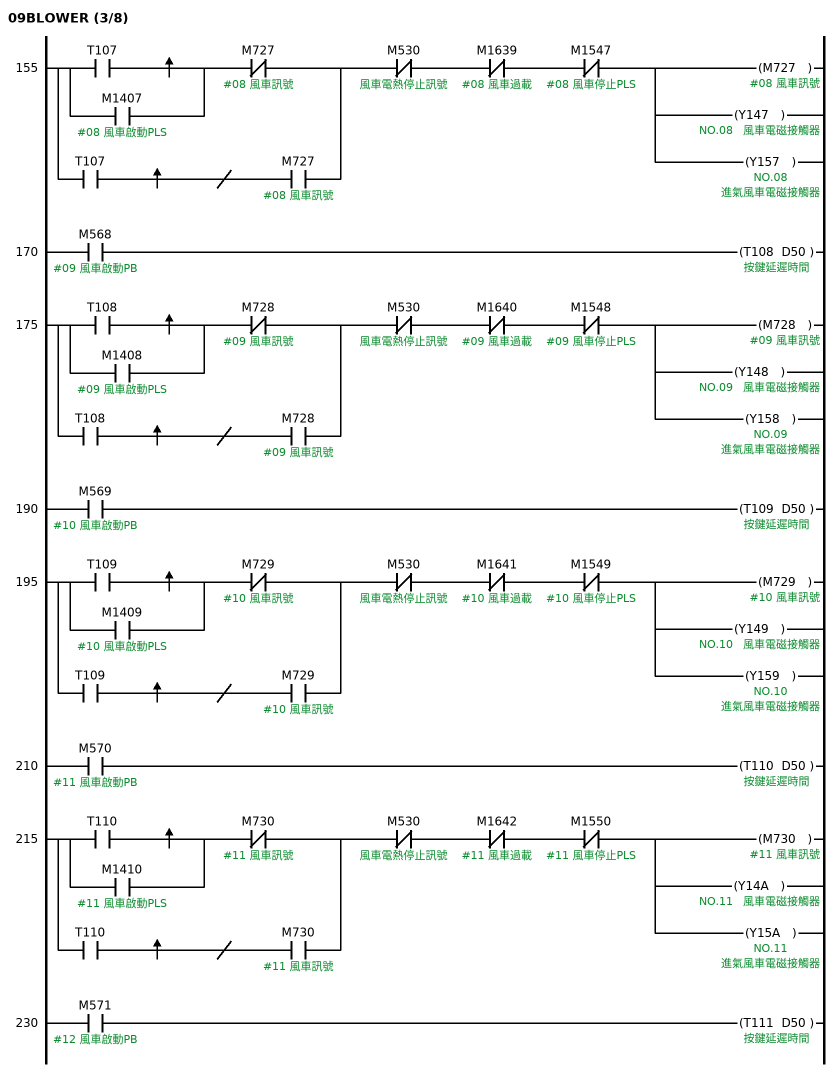
[picture p48: ladder of 09BLOWER, rungs at steps 155 to 230]
155   LD      T107
      MEP
      OR      M1407  ; #08 風車啟動PLS
      ANI     M727  ; #08 風車訊號
      LD      T107
      MEP
      INV
      AND     M727  ; #08 風車訊號
      ORB
      ANI     M530  ; 風車電熱停止訊號
      ANI     M1639  ; #08 風車過載
      ANI     M1547  ; #08 風車停止PLS
      OUT     M727  ; #08 風車訊號
      OUT     Y147  ; NO.08   風車電磁接觸器
      OUT     Y157  ; NO.08   進氣風車電磁接觸器
170   LD      M568  ; #09 風車啟動PB
      OUT     T108 D50  ; 按鍵延遲時間
175   LD      T108
      MEP
      OR      M1408  ; #09 風車啟動PLS
      ANI     M728  ; #09 風車訊號
      LD      T108
      MEP
      INV
      AND     M728  ; #09 風車訊號
      ORB
      ANI     M530  ; 風車電熱停止訊號
      ANI     M1640  ; #09 風車過載
      ANI     M1548  ; #09 風車停止PLS
      OUT     M728  ; #09 風車訊號
      OUT     Y148  ; NO.09   風車電磁接觸器
      OUT     Y158  ; NO.09   進氣風車電磁接觸器
190   LD      M569  ; #10 風車啟動PB
      OUT     T109 D50  ; 按鍵延遲時間
195   LD      T109
      MEP
      OR      M1409  ; #10 風車啟動PLS
      ANI     M729  ; #10 風車訊號
      LD      T109
      MEP
      INV
      AND     M729  ; #10 風車訊號
      ORB
      ANI     M530  ; 風車電熱停止訊號
      ANI     M1641  ; #10 風車過載
      ANI     M1549  ; #10 風車停止PLS
      OUT     M729  ; #10 風車訊號
      OUT     Y149  ; NO.10   風車電磁接觸器
      OUT     Y159  ; NO.10   進氣風車電磁接觸器
210   LD      M570  ; #11 風車啟動PB
      OUT     T110 D50  ; 按鍵延遲時間
215   LD      T110
      MEP
      OR      M1410  ; #11 風車啟動PLS
      ANI     M730  ; #11 風車訊號
      LD      T110
      MEP
      INV
      AND     M730  ; #11 風車訊號
      ORB
      ANI     M530  ; 風車電熱停止訊號
      ANI     M1642  ; #11 風車過載
      ANI     M1550  ; #11 風車停止PLS
      OUT     M730  ; #11 風車訊號
      OUT     Y14A  ; NO.11   風車電磁接觸器
      OUT     Y15A  ; NO.11   進氣風車電磁接觸器
230   LD      M571  ; #12 風車啟動PB
      OUT     T111 D50  ; 按鍵延遲時間
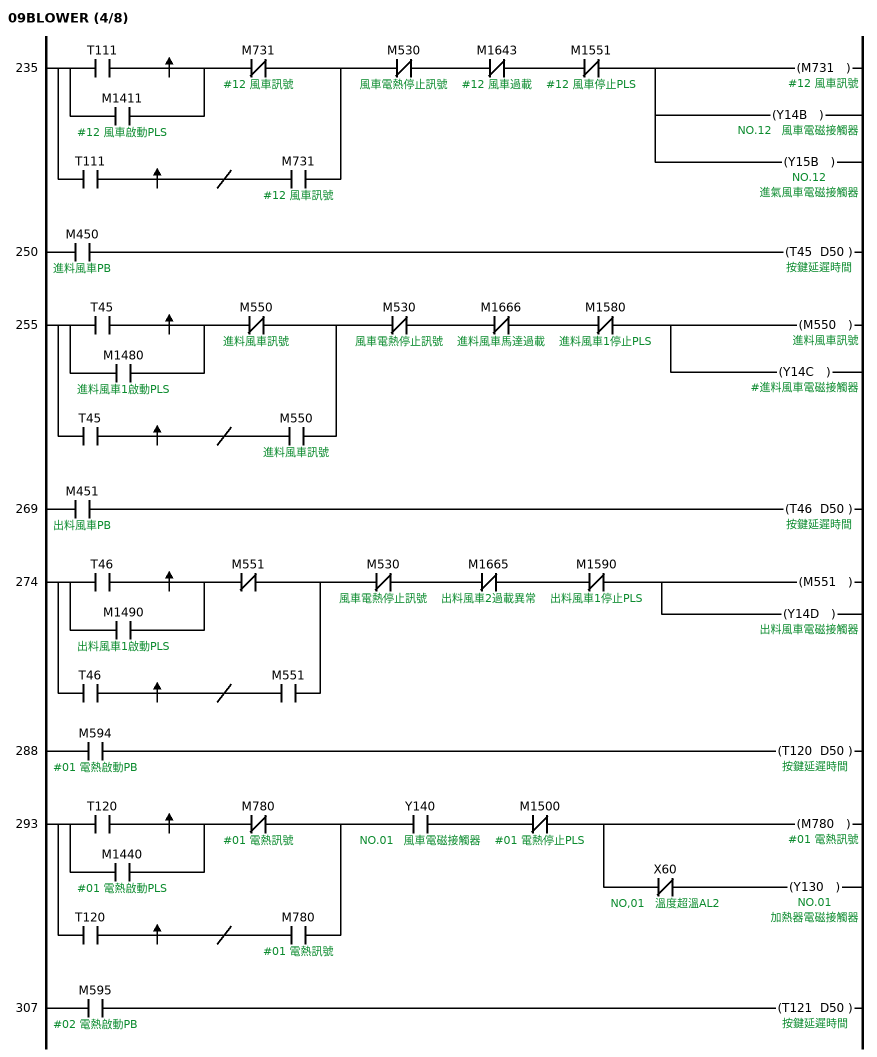
235   LD      T111
      MEP
      OR      M1411  ; #12 風車啟動PLS
      ANI     M731  ; #12 風車訊號
      LD      T111
      MEP
      INV
      AND     M731  ; #12 風車訊號
      ORB
      ANI     M530  ; 風車電熱停止訊號
      ANI     M1643  ; #12 風車過載
      ANI     M1551  ; #12 風車停止PLS
      OUT     M731  ; #12 風車訊號
      OUT     Y14B  ; NO.12   風車電磁接觸器
      OUT     Y15B  ; NO.12   進氣風車電磁接觸器
250   LD      M450  ; 進料風車PB
      OUT     T45 D50  ; 按鍵延遲時間
255   LD      T45
      MEP
      OR      M1480  ; 進料風車1啟動PLS
      ANI     M550  ; 進料風車訊號
      LD      T45
      MEP
      INV
      AND     M550  ; 進料風車訊號
      ORB
      ANI     M530  ; 風車電熱停止訊號
      ANI     M1666  ; 進料風車馬達過載
      ANI     M1580  ; 進料風車1停止PLS
      OUT     M550  ; 進料風車訊號
      OUT     Y14C  ; #進料風車電磁接觸器
269   LD      M451  ; 出料風車PB
      OUT     T46 D50  ; 按鍵延遲時間
274   LD      T46
      MEP
      OR      M1490  ; 出料風車1啟動PLS
      ANI     M551
      LD      T46
      MEP
      INV
      AND     M551
      ORB
      ANI     M530  ; 風車電熱停止訊號
      ANI     M1665  ; 出料風車2過載異常
      ANI     M1590  ; 出料風車1停止PLS
      OUT     M551
      OUT     Y14D  ; 出料風車電磁接觸器
288   LD      M594  ; #01 電熱啟動PB
      OUT     T120 D50  ; 按鍵延遲時間
293   LD      T120
      MEP
      OR      M1440  ; #01 電熱啟動PLS
      ANI     M780  ; #01 電熱訊號
      LD      T120
      MEP
      INV
      AND     M780  ; #01 電熱訊號
      ORB
      AND     Y140  ; NO.01   風車電磁接觸器
      ANI     M1500  ; #01 電熱停止PLS
      OUT     M780  ; #01 電熱訊號
      ANI     X60  ; NO,01   溫度超溫AL2
      OUT     Y130  ; NO.01   加熱器電磁接觸器
307   LD      M595  ; #02 電熱啟動PB
      OUT     T121 D50  ; 按鍵延遲時間
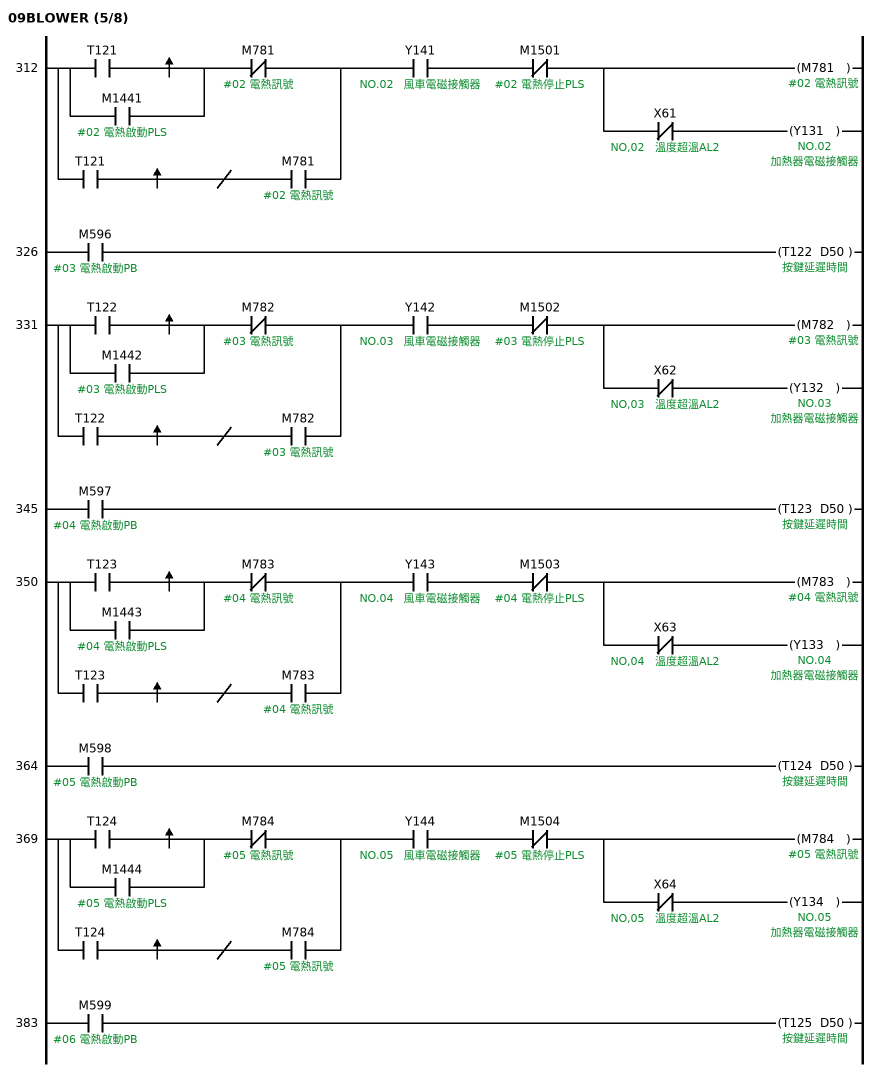
312   LD      T121
      MEP
      OR      M1441  ; #02 電熱啟動PLS
      ANI     M781  ; #02 電熱訊號
      LD      T121
      MEP
      INV
      AND     M781  ; #02 電熱訊號
      ORB
      AND     Y141  ; NO.02   風車電磁接觸器
      ANI     M1501  ; #02 電熱停止PLS
      OUT     M781  ; #02 電熱訊號
      ANI     X61  ; NO,02   溫度超溫AL2
      OUT     Y131  ; NO.02   加熱器電磁接觸器
326   LD      M596  ; #03 電熱啟動PB
      OUT     T122 D50  ; 按鍵延遲時間
331   LD      T122
      MEP
      OR      M1442  ; #03 電熱啟動PLS
      ANI     M782  ; #03 電熱訊號
      LD      T122
      MEP
      INV
      AND     M782  ; #03 電熱訊號
      ORB
      AND     Y142  ; NO.03   風車電磁接觸器
      ANI     M1502  ; #03 電熱停止PLS
      OUT     M782  ; #03 電熱訊號
      ANI     X62  ; NO,03   溫度超溫AL2
      OUT     Y132  ; NO.03   加熱器電磁接觸器
345   LD      M597  ; #04 電熱啟動PB
      OUT     T123 D50  ; 按鍵延遲時間
350   LD      T123
      MEP
      OR      M1443  ; #04 電熱啟動PLS
      ANI     M783  ; #04 電熱訊號
      LD      T123
      MEP
      INV
      AND     M783  ; #04 電熱訊號
      ORB
      AND     Y143  ; NO.04   風車電磁接觸器
      ANI     M1503  ; #04 電熱停止PLS
      OUT     M783  ; #04 電熱訊號
      ANI     X63  ; NO,04   溫度超溫AL2
      OUT     Y133  ; NO.04   加熱器電磁接觸器
364   LD      M598  ; #05 電熱啟動PB
      OUT     T124 D50  ; 按鍵延遲時間
369   LD      T124
      MEP
      OR      M1444  ; #05 電熱啟動PLS
      ANI     M784  ; #05 電熱訊號
      LD      T124
      MEP
      INV
      AND     M784  ; #05 電熱訊號
      ORB
      AND     Y144  ; NO.05   風車電磁接觸器
      ANI     M1504  ; #05 電熱停止PLS
      OUT     M784  ; #05 電熱訊號
      ANI     X64  ; NO,05   溫度超溫AL2
      OUT     Y134  ; NO.05   加熱器電磁接觸器
383   LD      M599  ; #06 電熱啟動PB
      OUT     T125 D50  ; 按鍵延遲時間
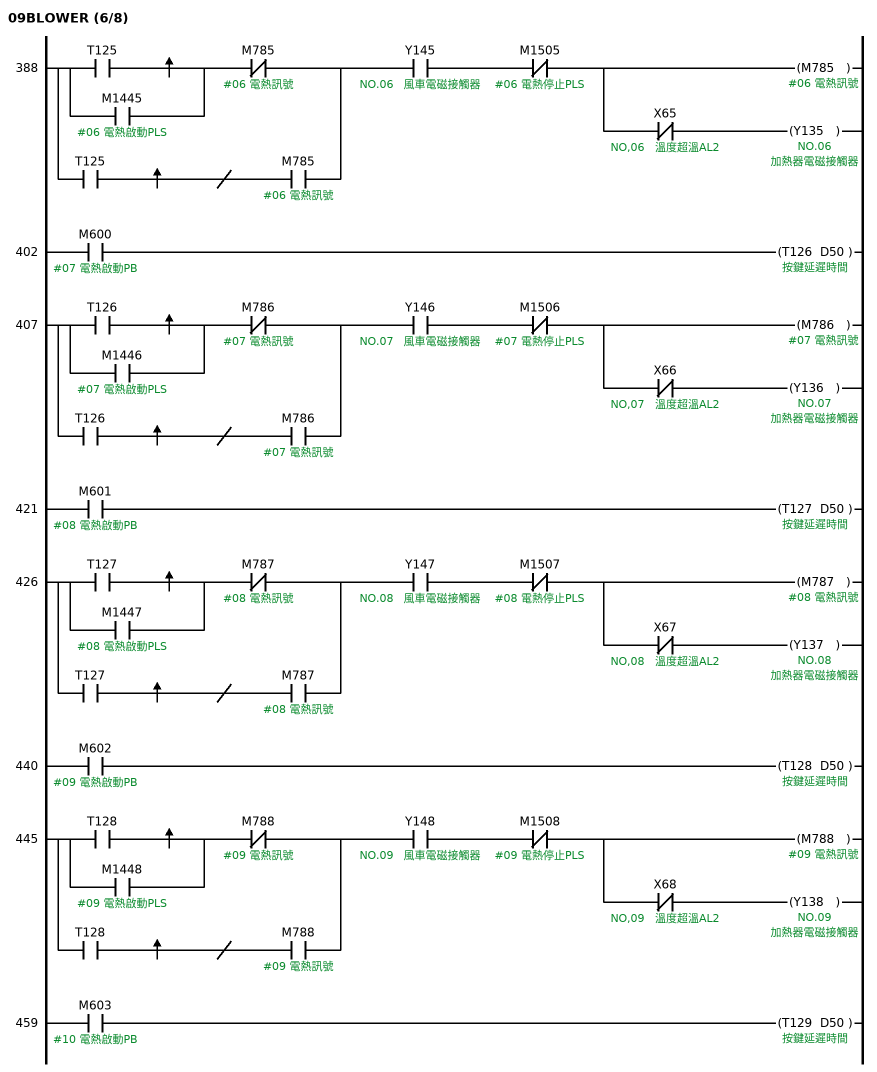
388   LD      T125
      MEP
      OR      M1445  ; #06 電熱啟動PLS
      ANI     M785  ; #06 電熱訊號
      LD      T125
      MEP
      INV
      AND     M785  ; #06 電熱訊號
      ORB
      AND     Y145  ; NO.06   風車電磁接觸器
      ANI     M1505  ; #06 電熱停止PLS
      OUT     M785  ; #06 電熱訊號
      ANI     X65  ; NO,06   溫度超溫AL2
      OUT     Y135  ; NO.06   加熱器電磁接觸器
402   LD      M600  ; #07 電熱啟動PB
      OUT     T126 D50  ; 按鍵延遲時間
407   LD      T126
      MEP
      OR      M1446  ; #07 電熱啟動PLS
      ANI     M786  ; #07 電熱訊號
      LD      T126
      MEP
      INV
      AND     M786  ; #07 電熱訊號
      ORB
      AND     Y146  ; NO.07   風車電磁接觸器
      ANI     M1506  ; #07 電熱停止PLS
      OUT     M786  ; #07 電熱訊號
      ANI     X66  ; NO,07   溫度超溫AL2
      OUT     Y136  ; NO.07   加熱器電磁接觸器
421   LD      M601  ; #08 電熱啟動PB
      OUT     T127 D50  ; 按鍵延遲時間
426   LD      T127
      MEP
      OR      M1447  ; #08 電熱啟動PLS
      ANI     M787  ; #08 電熱訊號
      LD      T127
      MEP
      INV
      AND     M787  ; #08 電熱訊號
      ORB
      AND     Y147  ; NO.08   風車電磁接觸器
      ANI     M1507  ; #08 電熱停止PLS
      OUT     M787  ; #08 電熱訊號
      ANI     X67  ; NO,08   溫度超溫AL2
      OUT     Y137  ; NO.08   加熱器電磁接觸器
440   LD      M602  ; #09 電熱啟動PB
      OUT     T128 D50  ; 按鍵延遲時間
445   LD      T128
      MEP
      OR      M1448  ; #09 電熱啟動PLS
      ANI     M788  ; #09 電熱訊號
      LD      T128
      MEP
      INV
      AND     M788  ; #09 電熱訊號
      ORB
      AND     Y148  ; NO.09   風車電磁接觸器
      ANI     M1508  ; #09 電熱停止PLS
      OUT     M788  ; #09 電熱訊號
      ANI     X68  ; NO,09   溫度超溫AL2
      OUT     Y138  ; NO.09   加熱器電磁接觸器
459   LD      M603  ; #10 電熱啟動PB
      OUT     T129 D50  ; 按鍵延遲時間
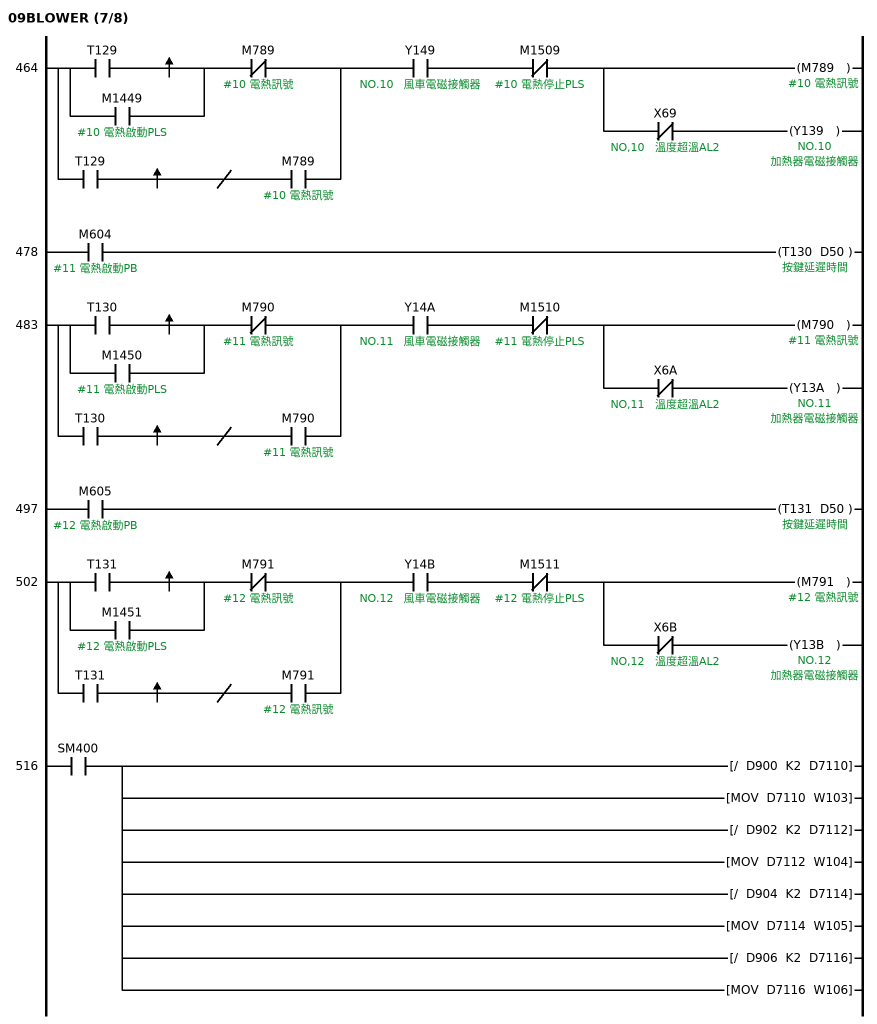
464   LD      T129
      MEP
      OR      M1449  ; #10 電熱啟動PLS
      ANI     M789  ; #10 電熱訊號
      LD      T129
      MEP
      INV
      AND     M789  ; #10 電熱訊號
      ORB
      AND     Y149  ; NO.10   風車電磁接觸器
      ANI     M1509  ; #10 電熱停止PLS
      OUT     M789  ; #10 電熱訊號
      ANI     X69  ; NO,10   溫度超溫AL2
      OUT     Y139  ; NO.10   加熱器電磁接觸器
478   LD      M604  ; #11 電熱啟動PB
      OUT     T130 D50  ; 按鍵延遲時間
483   LD      T130
      MEP
      OR      M1450  ; #11 電熱啟動PLS
      ANI     M790  ; #11 電熱訊號
      LD      T130
      MEP
      INV
      AND     M790  ; #11 電熱訊號
      ORB
      AND     Y14A  ; NO.11   風車電磁接觸器
      ANI     M1510  ; #11 電熱停止PLS
      OUT     M790  ; #11 電熱訊號
      ANI     X6A  ; NO,11   溫度超溫AL2
      OUT     Y13A  ; NO.11   加熱器電磁接觸器
497   LD      M605  ; #12 電熱啟動PB
      OUT     T131 D50  ; 按鍵延遲時間
502   LD      T131
      MEP
      OR      M1451  ; #12 電熱啟動PLS
      ANI     M791  ; #12 電熱訊號
      LD      T131
      MEP
      INV
      AND     M791  ; #12 電熱訊號
      ORB
      AND     Y14B  ; NO.12   風車電磁接觸器
      ANI     M1511  ; #12 電熱停止PLS
      OUT     M791  ; #12 電熱訊號
      ANI     X6B  ; NO,12   溫度超溫AL2
      OUT     Y13B  ; NO.12   加熱器電磁接觸器
516   LD      SM400
      /       D900 K2 D7110
      MOV     D7110 W103
      /       D902 K2 D7112
      MOV     D7112 W104
      /       D904 K2 D7114
      MOV     D7114 W105
      /       D906 K2 D7116
      MOV     D7116 W106
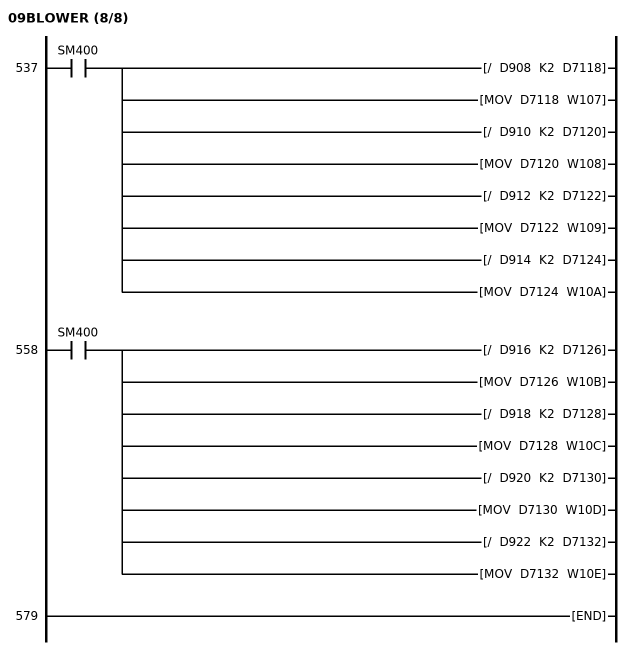
537   LD      SM400
      /       D908 K2 D7118
      MOV     D7118 W107
      /       D910 K2 D7120
      MOV     D7120 W108
      /       D912 K2 D7122
      MOV     D7122 W109
      /       D914 K2 D7124
      MOV     D7124 W10A
558   LD      SM400
      /       D916 K2 D7126
      MOV     D7126 W10B
      /       D918 K2 D7128
      MOV     D7128 W10C
      /       D920 K2 D7130
      MOV     D7130 W10D
      /       D922 K2 D7132
      MOV     D7132 W10E
579   END
END_PROGRAM

PROGRAM 10YIELD
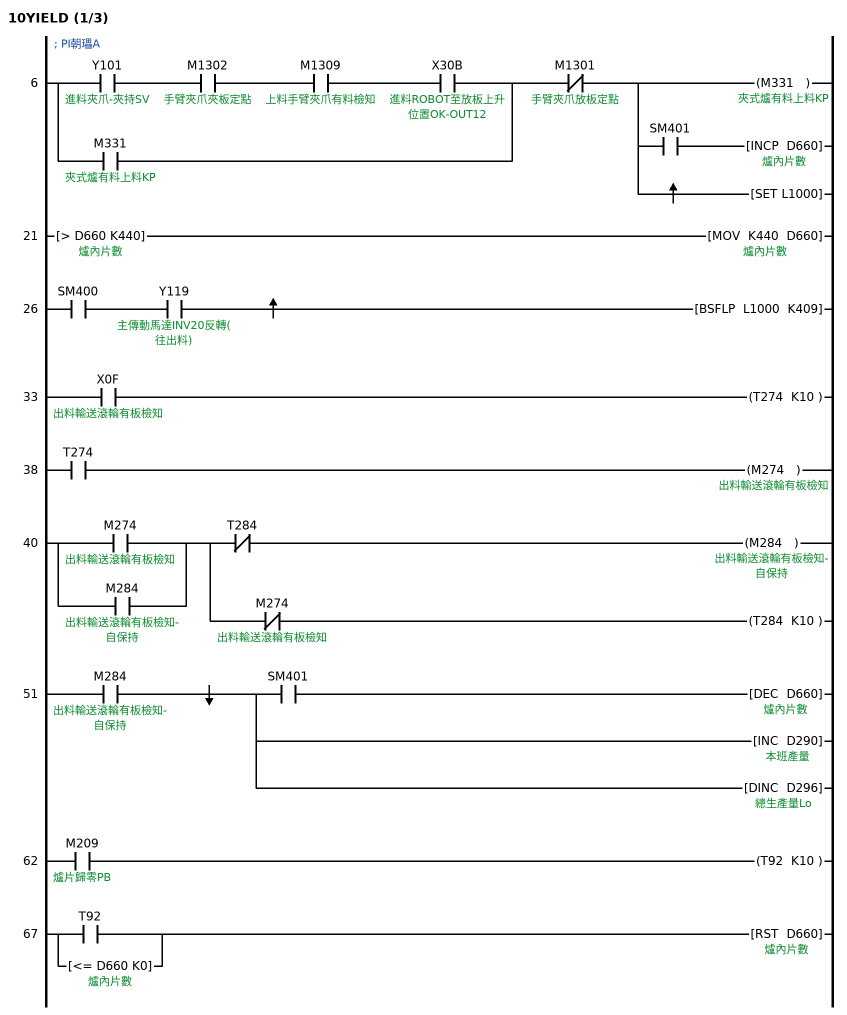
; PI朝瓃Α
6     LD      Y101  ; 進料夾爪-夾持SV
      AND     M1302  ; 手臂夾爪夾板定點
      AND     M1309  ; 上料手臂夾爪有料檢知
      AND     X30B  ; 進料ROBOT至放板上升位置OK-OUT12
      OR      M331  ; 夾式爐有料上料KP
      ANI     M1301  ; 手臂夾爪放板定點
      OUT     M331  ; 夾式爐有料上料KP
      MPS
      AND     SM401
      INCP    D660  ; 爐內片數
      MPP
      MEP
      SET     L1000
21    LD>     D660 K440  ; 爐內片數
      MOV     K440 D660
26    LD      SM400
      AND     Y119  ; 主傳動馬達INV20反轉(往出料)
      MEP
      BSFLP   L1000 K409
33    LD      X0F  ; 出料輸送滾輪有板檢知
      OUT     T274 K10
38    LD      T274
      OUT     M274  ; 出料輸送滾輪有板檢知
40    LD      M274  ; 出料輸送滾輪有板檢知
      OR      M284  ; 出料輸送滾輪有板檢知-自保持
      MPS
      ANI     T284
      OUT     M284  ; 出料輸送滾輪有板檢知-自保持
      MPP
      ANI     M274  ; 出料輸送滾輪有板檢知
      OUT     T284 K10
51    LD      M284  ; 出料輸送滾輪有板檢知-自保持
      MEF
      MPS
      AND     SM401
      DEC     D660
      MPP
      INC     D290  ; 本班產量
      DINC    D296  ; 總生產量Lo
62    LD      M209  ; 爐片歸零PB
      OUT     T92 K10
67    LD      T92
      OR<=    D660 K0  ; 爐內片數
      RST     D660  ; 爐內片數
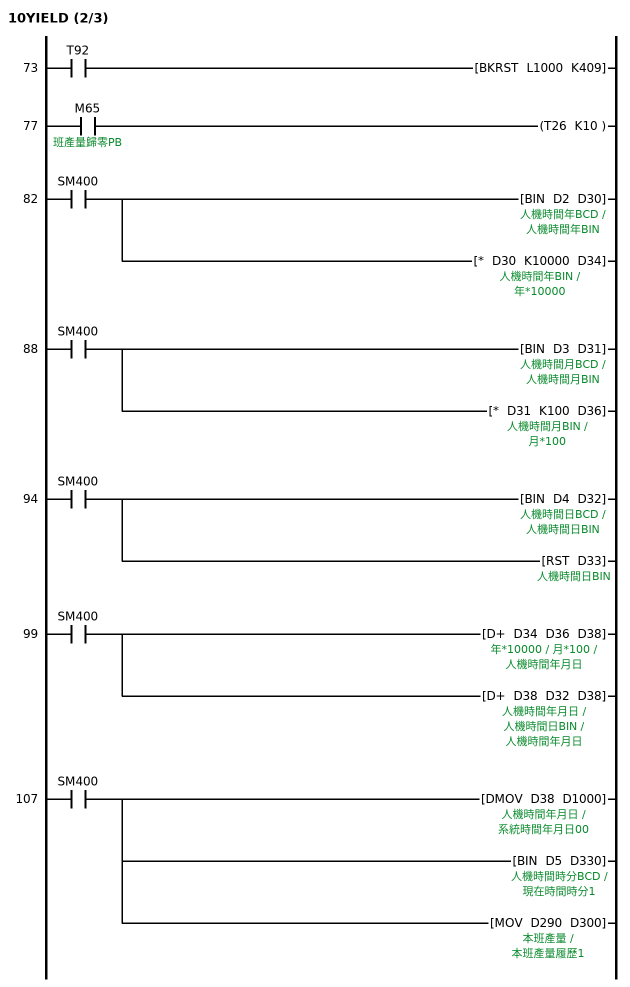
73    LD      T92
      BKRST   L1000 K409
77    LD      M65  ; 班產量歸零PB
      OUT     T26 K10
82    LD      SM400
      BIN     D2 D30  ; 人機時間年BCD / 人機時間年BIN
      *       D30 K10000 D34  ; 年*10000
88    LD      SM400
      BIN     D3 D31  ; 人機時間月BCD / 人機時間月BIN
      *       D31 K100 D36  ; 月*100
94    LD      SM400
      BIN     D4 D32  ; 人機時間日BCD / 人機時間日BIN
      RST     D33  ; 人機時間日BIN
99    LD      SM400
      D+      D34 D36 D38  ; 人機時間年月日
      D+      D38 D32 D38
107   LD      SM400
      DMOV    D38 D1000  ; 系統時間年月日00
      BIN     D5 D330  ; 人機時間時分BCD / 現在時間時分1
      MOV     D290 D300  ; 本班產量履歷1
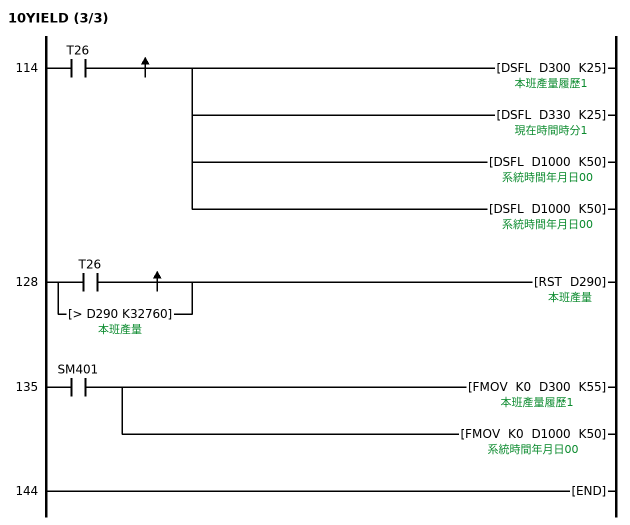
114   LD      T26
      MEP
      DSFL    D300 K25
      DSFL    D330 K25
      DSFL    D1000 K50
      DSFL    D1000 K50
128   LD      T26
      MEP
      OR>     D290 K32760  ; 本班產量
      RST     D290  ; 本班產量
135   LD      SM401
      FMOV    K0 D300 K55
      FMOV    K0 D1000 K50
144   END
END_PROGRAM

PROGRAM 11MAINTE
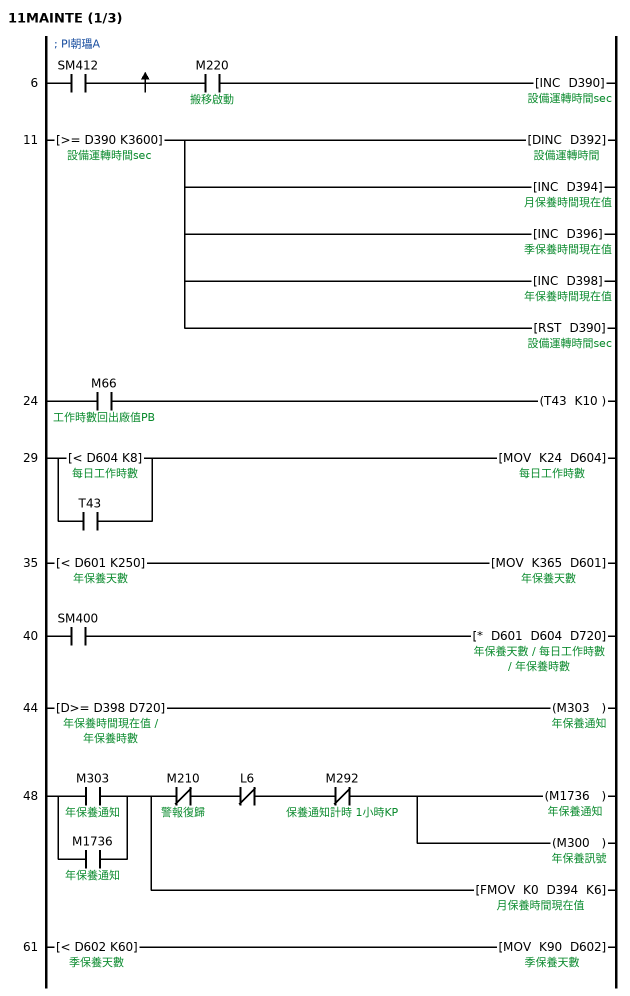
; PI朝瓃Α
6     LD      SM412
      MEP
      AND     M220  ; 搬移啟動
      INC     D390  ; 設備運轉時間sec
11    LD>=    D390 K3600  ; 設備運轉時間sec
      DINC    D392  ; 設備運轉時間
      INC     D394  ; 月保養時間現在值
      INC     D396  ; 季保養時間現在值
      INC     D398  ; 年保養時間現在值
      RST     D390  ; 設備運轉時間sec
24    LD      M66  ; 工作時數回出廠值PB
      OUT     T43 K10
29    LD<     D604 K8  ; 每日工作時數
      OR      T43
      MOV     K24 D604
35    LD<     D601 K250  ; 年保養天數
      MOV     K365 D601
40    LD      SM400
      *       D601 D604 D720  ; 年保養時數
44    LDD>=   D398 D720  ; 年保養時間現在值 / 年保養時數
      OUT     M303  ; 年保養通知
48    LD      M303  ; 年保養通知
      OR      M1736  ; 年保養通知
      MPS
      ANI     M210  ; 警報復歸
      ANI     L6
      ANI     M292  ; 保養通知計時 1小時KP
      OUT     M1736  ; 年保養通知
      OUT     M300  ; 年保養訊號
      MPP
      FMOV    K0 D394 K6
61    LD<     D602 K60  ; 季保養天數
      MOV     K90 D602
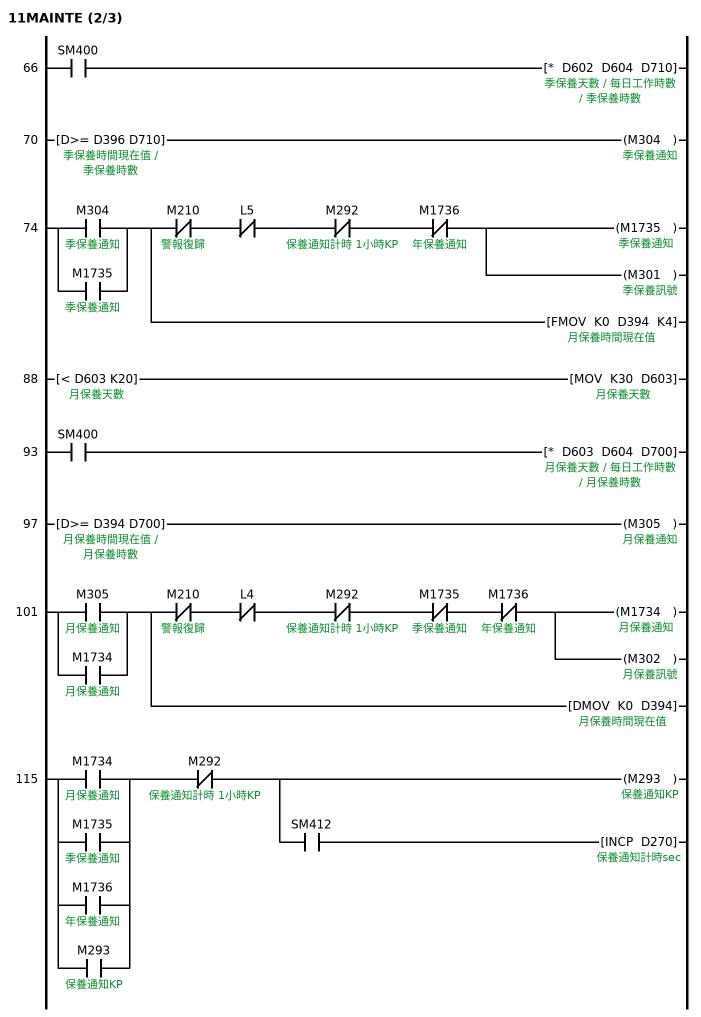
66    LD      SM400
      *       D602 D604 D710  ; 季保養時數
70    LDD>=   D396 D710  ; 季保養時間現在值 / 季保養時數
      OUT     M304  ; 季保養通知
74    LD      M304  ; 季保養通知
      OR      M1735  ; 季保養通知
      MPS
      ANI     M210  ; 警報復歸
      ANI     L5
      ANI     M292  ; 保養通知計時 1小時KP
      ANI     M1736  ; 年保養通知
      OUT     M1735  ; 季保養通知
      OUT     M301  ; 季保養訊號
      MPP
      FMOV    K0 D394 K4
88    LD<     D603 K20  ; 月保養天數
      MOV     K30 D603
93    LD      SM400
      *       D603 D604 D700  ; 月保養時數
97    LDD>=   D394 D700  ; 月保養時間現在值 / 月保養時數
      OUT     M305  ; 月保養通知
101   LD      M305  ; 月保養通知
      OR      M1734  ; 月保養通知
      MPS
      ANI     M210  ; 警報復歸
      ANI     L4
      ANI     M292  ; 保養通知計時 1小時KP
      ANI     M1735  ; 季保養通知
      ANI     M1736  ; 年保養通知
      OUT     M1734  ; 月保養通知
      OUT     M302  ; 月保養訊號
      MPP
      DMOV    K0 D394
115   LD      M1734  ; 月保養通知
      OR      M1735  ; 季保養通知
      OR      M1736  ; 年保養通知
      OR      M293  ; 保養通知KP
      ANI     M292  ; 保養通知計時 1小時KP
      OUT     M293  ; 保養通知KP
      AND     SM412
      INCP    D270  ; 保養通知計時sec
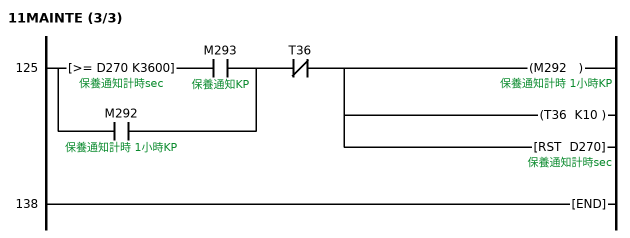
125   LD>=    D270 K3600  ; 保養通知計時sec
      AND     M293  ; 保養通知KP
      OR      M292  ; 保養通知計時 1小時KP
      ANI     T36
      OUT     M292  ; 保養通知計時 1小時KP
      OUT     T36 K10
      RST     D270  ; 保養通知計時sec
138   END
END_PROGRAM

PROGRAM 12ALARM1
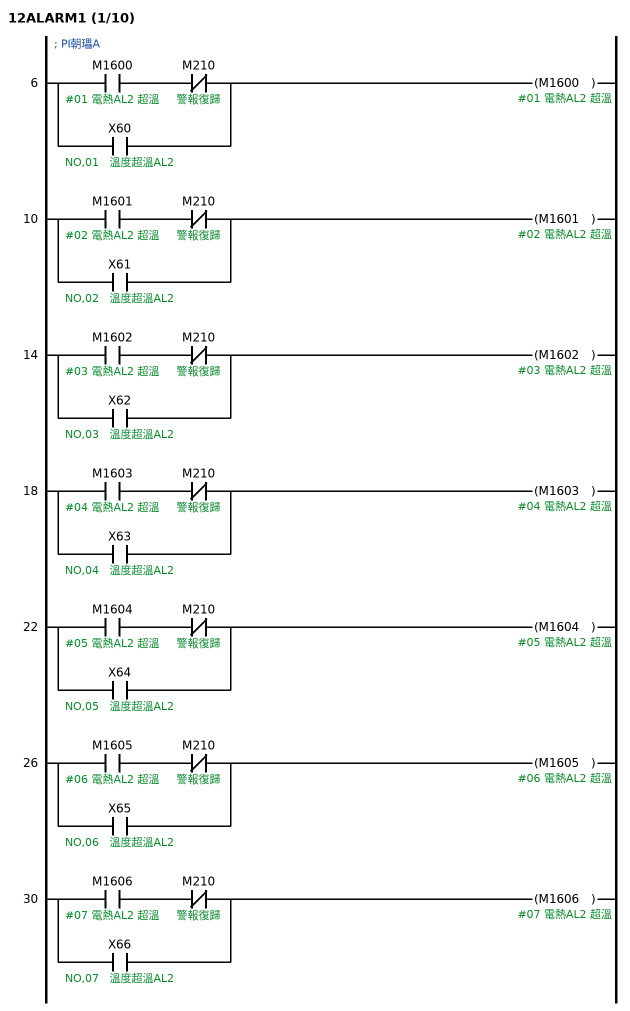
; PI朝瓃Α
6     LD      M1600  ; #01 電熱AL2 超溫
      ANI     M210  ; 警報復歸
      OR      X60  ; NO,01   溫度超溫AL2
      OUT     M1600  ; #01 電熱AL2 超溫
10    LD      M1601  ; #02 電熱AL2 超溫
      ANI     M210  ; 警報復歸
      OR      X61  ; NO,02   溫度超溫AL2
      OUT     M1601  ; #02 電熱AL2 超溫
14    LD      M1602  ; #03 電熱AL2 超溫
      ANI     M210  ; 警報復歸
      OR      X62  ; NO,03   溫度超溫AL2
      OUT     M1602  ; #03 電熱AL2 超溫
18    LD      M1603  ; #04 電熱AL2 超溫
      ANI     M210  ; 警報復歸
      OR      X63  ; NO,04   溫度超溫AL2
      OUT     M1603  ; #04 電熱AL2 超溫
22    LD      M1604  ; #05 電熱AL2 超溫
      ANI     M210  ; 警報復歸
      OR      X64  ; NO,05   溫度超溫AL2
      OUT     M1604  ; #05 電熱AL2 超溫
26    LD      M1605  ; #06 電熱AL2 超溫
      ANI     M210  ; 警報復歸
      OR      X65  ; NO,06   溫度超溫AL2
      OUT     M1605  ; #06 電熱AL2 超溫
30    LD      M1606  ; #07 電熱AL2 超溫
      ANI     M210  ; 警報復歸
      OR      X66  ; NO,07   溫度超溫AL2
      OUT     M1606  ; #07 電熱AL2 超溫
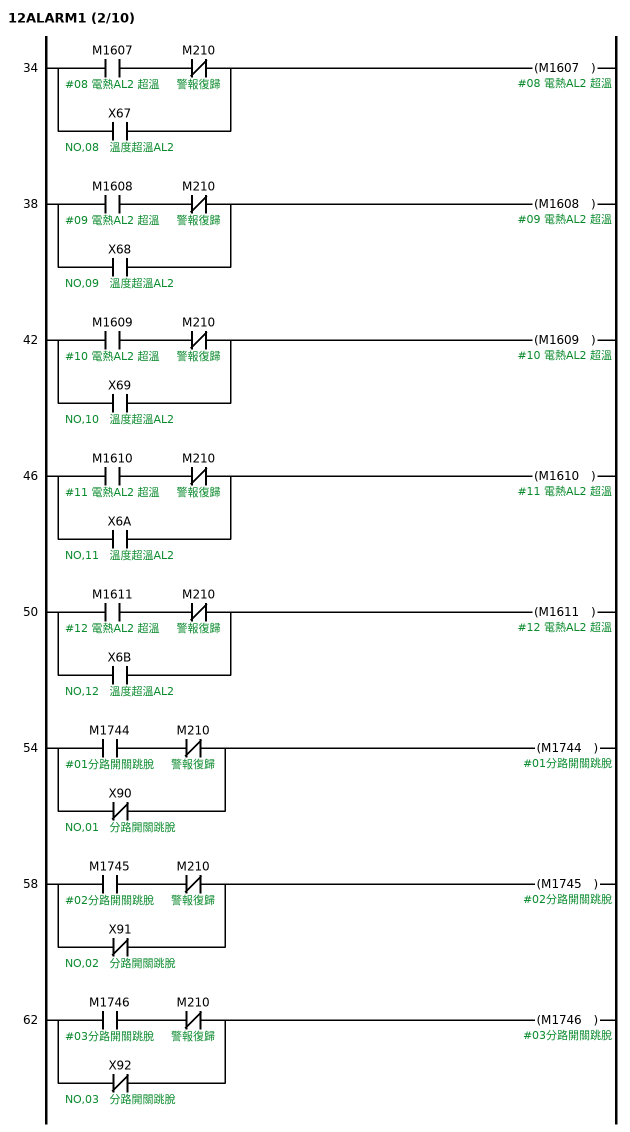
34    LD      M1607  ; #08 電熱AL2 超溫
      ANI     M210  ; 警報復歸
      OR      X67  ; NO,08   溫度超溫AL2
      OUT     M1607  ; #08 電熱AL2 超溫
38    LD      M1608  ; #09 電熱AL2 超溫
      ANI     M210  ; 警報復歸
      OR      X68  ; NO,09   溫度超溫AL2
      OUT     M1608  ; #09 電熱AL2 超溫
42    LD      M1609  ; #10 電熱AL2 超溫
      ANI     M210  ; 警報復歸
      OR      X69  ; NO,10   溫度超溫AL2
      OUT     M1609  ; #10 電熱AL2 超溫
46    LD      M1610  ; #11 電熱AL2 超溫
      ANI     M210  ; 警報復歸
      OR      X6A  ; NO,11   溫度超溫AL2
      OUT     M1610  ; #11 電熱AL2 超溫
50    LD      M1611  ; #12 電熱AL2 超溫
      ANI     M210  ; 警報復歸
      OR      X6B  ; NO,12   溫度超溫AL2
      OUT     M1611  ; #12 電熱AL2 超溫
54    LD      M1744  ; #01分路開關跳脫
      ANI     M210  ; 警報復歸
      ORI     X90  ; NO,01   分路開關跳脫
      OUT     M1744  ; #01分路開關跳脫
58    LD      M1745  ; #02分路開關跳脫
      ANI     M210  ; 警報復歸
      ORI     X91  ; NO,02   分路開關跳脫
      OUT     M1745  ; #02分路開關跳脫
62    LD      M1746  ; #03分路開關跳脫
      ANI     M210  ; 警報復歸
      ORI     X92  ; NO,03   分路開關跳脫
      OUT     M1746  ; #03分路開關跳脫
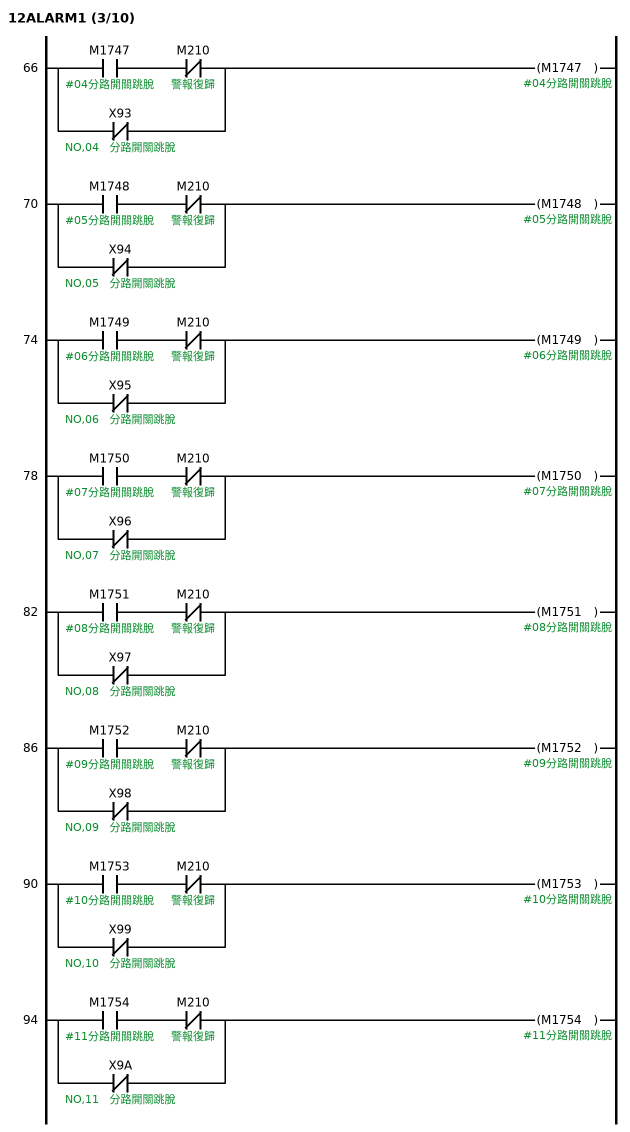
66    LD      M1747  ; #04分路開關跳脫
      ANI     M210  ; 警報復歸
      ORI     X93  ; NO,04   分路開關跳脫
      OUT     M1747  ; #04分路開關跳脫
70    LD      M1748  ; #05分路開關跳脫
      ANI     M210  ; 警報復歸
      ORI     X94  ; NO,05   分路開關跳脫
      OUT     M1748  ; #05分路開關跳脫
74    LD      M1749  ; #06分路開關跳脫
      ANI     M210  ; 警報復歸
      ORI     X95  ; NO,06   分路開關跳脫
      OUT     M1749  ; #06分路開關跳脫
78    LD      M1750  ; #07分路開關跳脫
      ANI     M210  ; 警報復歸
      ORI     X96  ; NO,07   分路開關跳脫
      OUT     M1750  ; #07分路開關跳脫
82    LD      M1751  ; #08分路開關跳脫
      ANI     M210  ; 警報復歸
      ORI     X97  ; NO,08   分路開關跳脫
      OUT     M1751  ; #08分路開關跳脫
86    LD      M1752  ; #09分路開關跳脫
      ANI     M210  ; 警報復歸
      ORI     X98  ; NO,09   分路開關跳脫
      OUT     M1752  ; #09分路開關跳脫
90    LD      M1753  ; #10分路開關跳脫
      ANI     M210  ; 警報復歸
      ORI     X99  ; NO,10   分路開關跳脫
      OUT     M1753  ; #10分路開關跳脫
94    LD      M1754  ; #11分路開關跳脫
      ANI     M210  ; 警報復歸
      ORI     X9A  ; NO,11   分路開關跳脫
      OUT     M1754  ; #11分路開關跳脫
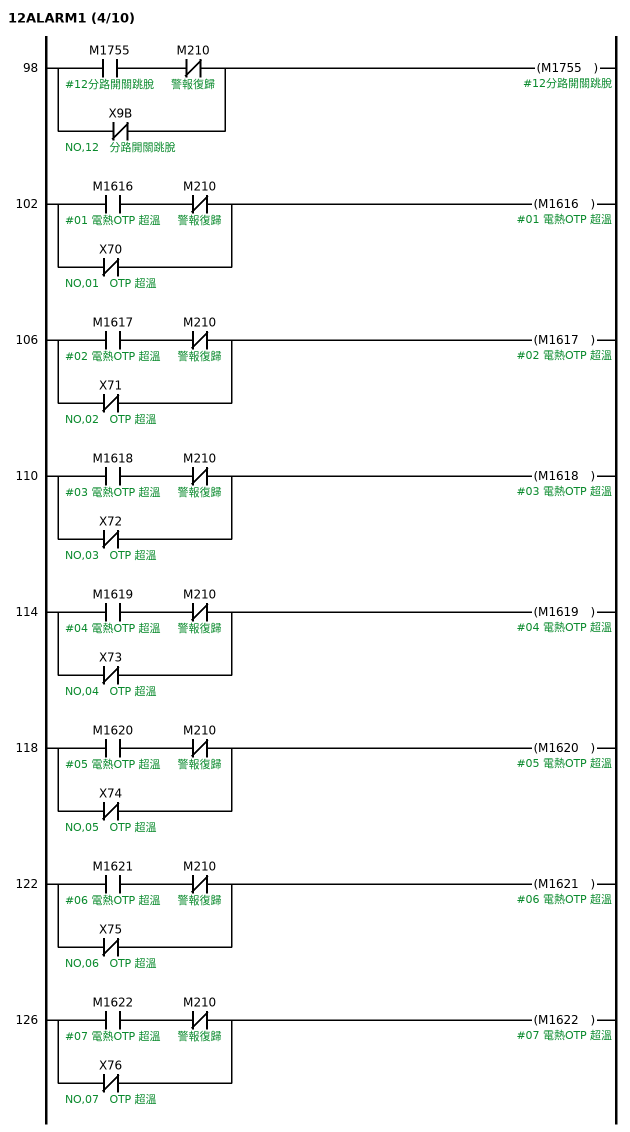
98    LD      M1755  ; #12分路開關跳脫
      ANI     M210  ; 警報復歸
      ORI     X9B  ; NO,12   分路開關跳脫
      OUT     M1755  ; #12分路開關跳脫
102   LD      M1616  ; #01 電熱OTP 超溫
      ANI     M210  ; 警報復歸
      ORI     X70  ; NO,01   OTP 超溫
      OUT     M1616  ; #01 電熱OTP 超溫
106   LD      M1617  ; #02 電熱OTP 超溫
      ANI     M210  ; 警報復歸
      ORI     X71  ; NO,02   OTP 超溫
      OUT     M1617  ; #02 電熱OTP 超溫
110   LD      M1618  ; #03 電熱OTP 超溫
      ANI     M210  ; 警報復歸
      ORI     X72  ; NO,03   OTP 超溫
      OUT     M1618  ; #03 電熱OTP 超溫
114   LD      M1619  ; #04 電熱OTP 超溫
      ANI     M210  ; 警報復歸
      ORI     X73  ; NO,04   OTP 超溫
      OUT     M1619  ; #04 電熱OTP 超溫
118   LD      M1620  ; #05 電熱OTP 超溫
      ANI     M210  ; 警報復歸
      ORI     X74  ; NO,05   OTP 超溫
      OUT     M1620  ; #05 電熱OTP 超溫
122   LD      M1621  ; #06 電熱OTP 超溫
      ANI     M210  ; 警報復歸
      ORI     X75  ; NO,06   OTP 超溫
      OUT     M1621  ; #06 電熱OTP 超溫
126   LD      M1622  ; #07 電熱OTP 超溫
      ANI     M210  ; 警報復歸
      ORI     X76  ; NO,07   OTP 超溫
      OUT     M1622  ; #07 電熱OTP 超溫
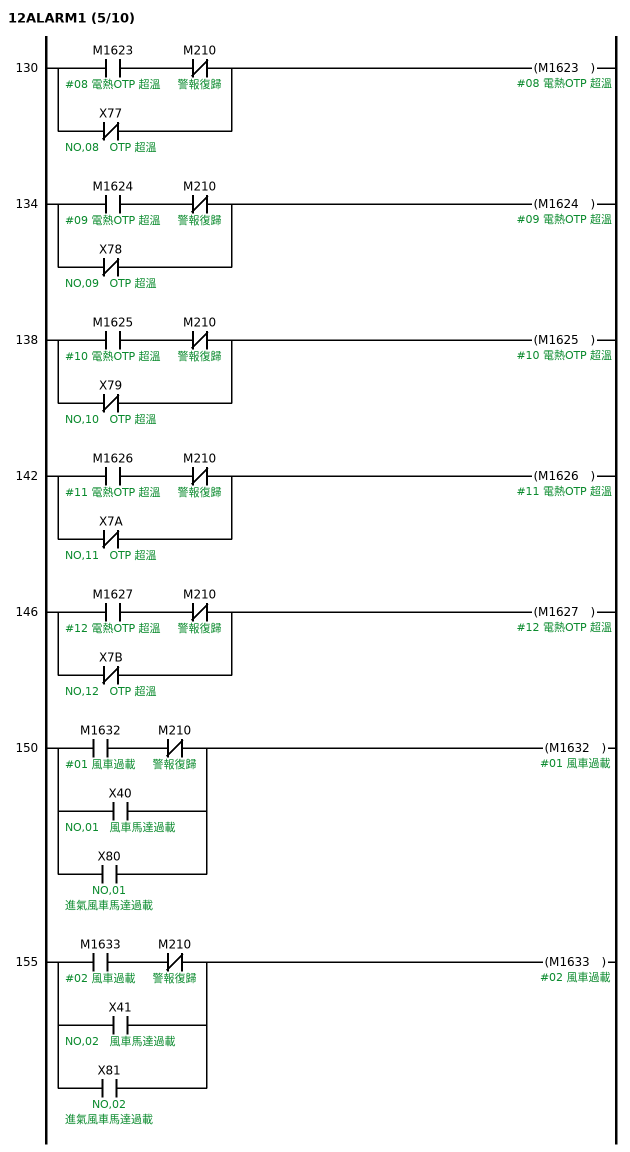
130   LD      M1623  ; #08 電熱OTP 超溫
      ANI     M210  ; 警報復歸
      ORI     X77  ; NO,08   OTP 超溫
      OUT     M1623  ; #08 電熱OTP 超溫
134   LD      M1624  ; #09 電熱OTP 超溫
      ANI     M210  ; 警報復歸
      ORI     X78  ; NO,09   OTP 超溫
      OUT     M1624  ; #09 電熱OTP 超溫
138   LD      M1625  ; #10 電熱OTP 超溫
      ANI     M210  ; 警報復歸
      ORI     X79  ; NO,10   OTP 超溫
      OUT     M1625  ; #10 電熱OTP 超溫
142   LD      M1626  ; #11 電熱OTP 超溫
      ANI     M210  ; 警報復歸
      ORI     X7A  ; NO,11   OTP 超溫
      OUT     M1626  ; #11 電熱OTP 超溫
146   LD      M1627  ; #12 電熱OTP 超溫
      ANI     M210  ; 警報復歸
      ORI     X7B  ; NO,12   OTP 超溫
      OUT     M1627  ; #12 電熱OTP 超溫
150   LD      M1632  ; #01 風車過載
      ANI     M210  ; 警報復歸
      OR      X40  ; NO,01   風車馬達過載
      OR      X80  ; NO,01   進氣風車馬達過載
      OUT     M1632  ; #01 風車過載
155   LD      M1633  ; #02 風車過載
      ANI     M210  ; 警報復歸
      OR      X41  ; NO,02   風車馬達過載
      OR      X81  ; NO,02   進氣風車馬達過載
      OUT     M1633  ; #02 風車過載
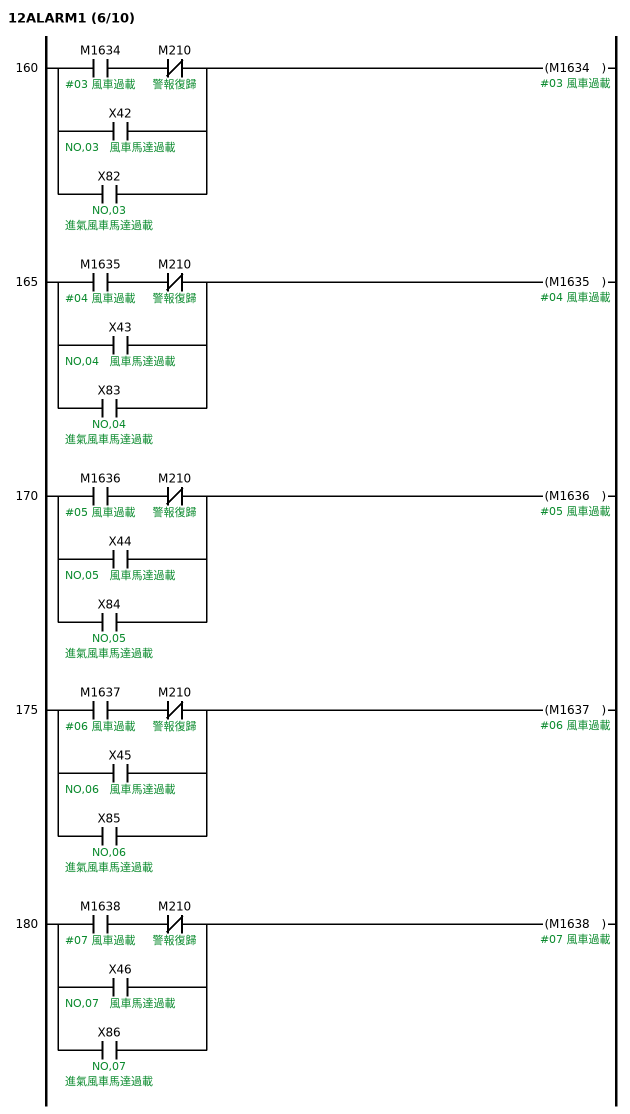
160   LD      M1634  ; #03 風車過載
      ANI     M210  ; 警報復歸
      OR      X42  ; NO,03   風車馬達過載
      OR      X82  ; NO,03   進氣風車馬達過載
      OUT     M1634  ; #03 風車過載
165   LD      M1635  ; #04 風車過載
      ANI     M210  ; 警報復歸
      OR      X43  ; NO,04   風車馬達過載
      OR      X83  ; NO,04   進氣風車馬達過載
      OUT     M1635  ; #04 風車過載
170   LD      M1636  ; #05 風車過載
      ANI     M210  ; 警報復歸
      OR      X44  ; NO,05   風車馬達過載
      OR      X84  ; NO,05   進氣風車馬達過載
      OUT     M1636  ; #05 風車過載
175   LD      M1637  ; #06 風車過載
      ANI     M210  ; 警報復歸
      OR      X45  ; NO,06   風車馬達過載
      OR      X85  ; NO,06   進氣風車馬達過載
      OUT     M1637  ; #06 風車過載
180   LD      M1638  ; #07 風車過載
      ANI     M210  ; 警報復歸
      OR      X46  ; NO,07   風車馬達過載
      OR      X86  ; NO,07   進氣風車馬達過載
      OUT     M1638  ; #07 風車過載
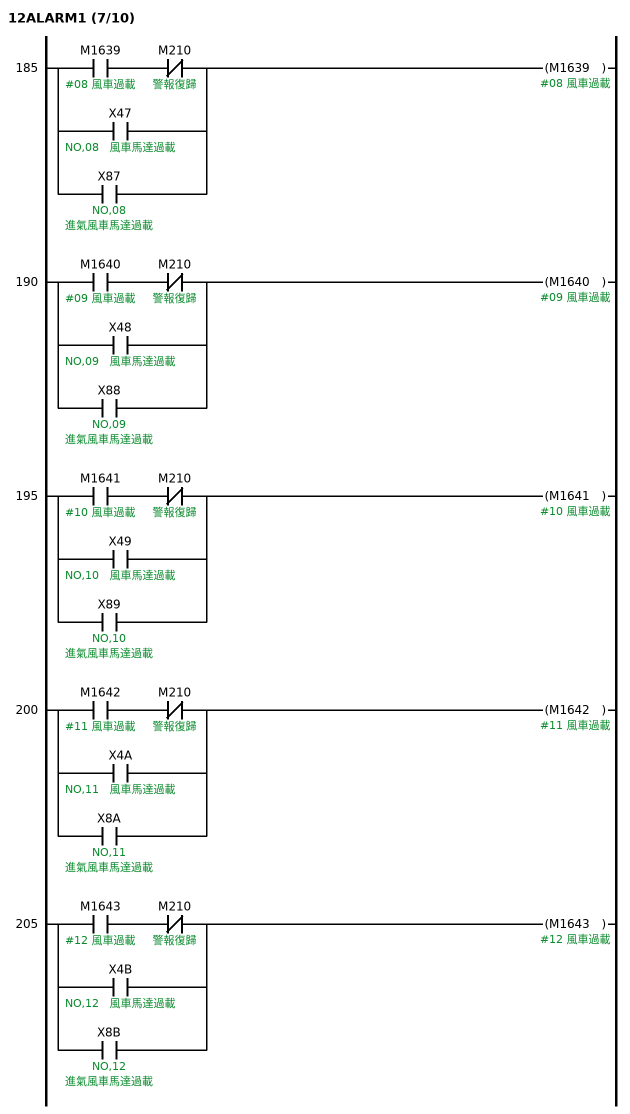
185   LD      M1639  ; #08 風車過載
      ANI     M210  ; 警報復歸
      OR      X47  ; NO,08   風車馬達過載
      OR      X87  ; NO,08   進氣風車馬達過載
      OUT     M1639  ; #08 風車過載
190   LD      M1640  ; #09 風車過載
      ANI     M210  ; 警報復歸
      OR      X48  ; NO,09   風車馬達過載
      OR      X88  ; NO,09   進氣風車馬達過載
      OUT     M1640  ; #09 風車過載
195   LD      M1641  ; #10 風車過載
      ANI     M210  ; 警報復歸
      OR      X49  ; NO,10   風車馬達過載
      OR      X89  ; NO,10   進氣風車馬達過載
      OUT     M1641  ; #10 風車過載
200   LD      M1642  ; #11 風車過載
      ANI     M210  ; 警報復歸
      OR      X4A  ; NO,11   風車馬達過載
      OR      X8A  ; NO,11   進氣風車馬達過載
      OUT     M1642  ; #11 風車過載
205   LD      M1643  ; #12 風車過載
      ANI     M210  ; 警報復歸
      OR      X4B  ; NO,12   風車馬達過載
      OR      X8B  ; NO,12   進氣風車馬達過載
      OUT     M1643  ; #12 風車過載
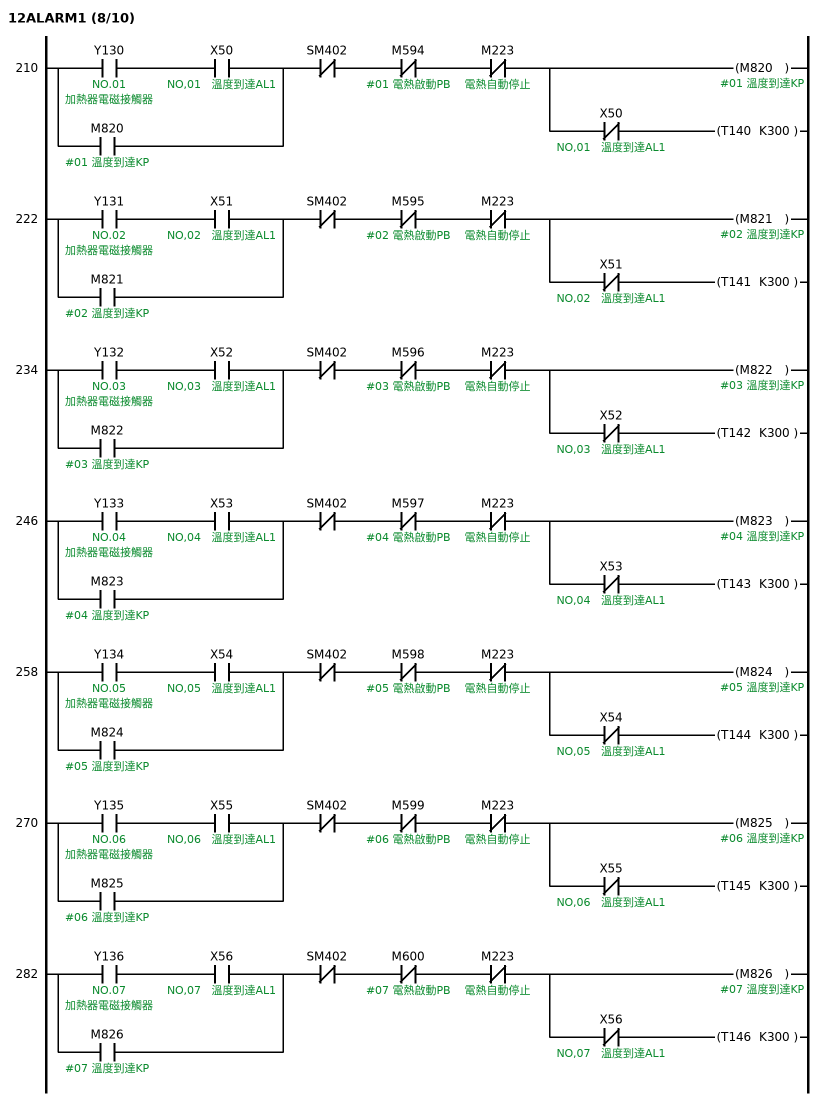
210   LD      Y130  ; NO.01   加熱器電磁接觸器
      AND     X50  ; NO,01   溫度到達AL1
      OR      M820  ; #01 溫度到達KP
      ANI     SM402
      ANI     M594  ; #01 電熱啟動PB
      ANI     M223  ; 電熱自動停止
      OUT     M820  ; #01 溫度到達KP
      ANI     X50  ; NO,01   溫度到達AL1
      OUT     T140 K300
222   LD      Y131  ; NO.02   加熱器電磁接觸器
      AND     X51  ; NO,02   溫度到達AL1
      OR      M821  ; #02 溫度到達KP
      ANI     SM402
      ANI     M595  ; #02 電熱啟動PB
      ANI     M223  ; 電熱自動停止
      OUT     M821  ; #02 溫度到達KP
      ANI     X51  ; NO,02   溫度到達AL1
      OUT     T141 K300
234   LD      Y132  ; NO.03   加熱器電磁接觸器
      AND     X52  ; NO,03   溫度到達AL1
      OR      M822  ; #03 溫度到達KP
      ANI     SM402
      ANI     M596  ; #03 電熱啟動PB
      ANI     M223  ; 電熱自動停止
      OUT     M822  ; #03 溫度到達KP
      ANI     X52  ; NO,03   溫度到達AL1
      OUT     T142 K300
246   LD      Y133  ; NO.04   加熱器電磁接觸器
      AND     X53  ; NO,04   溫度到達AL1
      OR      M823  ; #04 溫度到達KP
      ANI     SM402
      ANI     M597  ; #04 電熱啟動PB
      ANI     M223  ; 電熱自動停止
      OUT     M823  ; #04 溫度到達KP
      ANI     X53  ; NO,04   溫度到達AL1
      OUT     T143 K300
258   LD      Y134  ; NO.05   加熱器電磁接觸器
      AND     X54  ; NO,05   溫度到達AL1
      OR      M824  ; #05 溫度到達KP
      ANI     SM402
      ANI     M598  ; #05 電熱啟動PB
      ANI     M223  ; 電熱自動停止
      OUT     M824  ; #05 溫度到達KP
      ANI     X54  ; NO,05   溫度到達AL1
      OUT     T144 K300
270   LD      Y135  ; NO.06   加熱器電磁接觸器
      AND     X55  ; NO,06   溫度到達AL1
      OR      M825  ; #06 溫度到達KP
      ANI     SM402
      ANI     M599  ; #06 電熱啟動PB
      ANI     M223  ; 電熱自動停止
      OUT     M825  ; #06 溫度到達KP
      ANI     X55  ; NO,06   溫度到達AL1
      OUT     T145 K300
282   LD      Y136  ; NO.07   加熱器電磁接觸器
      AND     X56  ; NO,07   溫度到達AL1
      OR      M826  ; #07 溫度到達KP
      ANI     SM402
      ANI     M600  ; #07 電熱啟動PB
      ANI     M223  ; 電熱自動停止
      OUT     M826  ; #07 溫度到達KP
      ANI     X56  ; NO,07   溫度到達AL1
      OUT     T146 K300
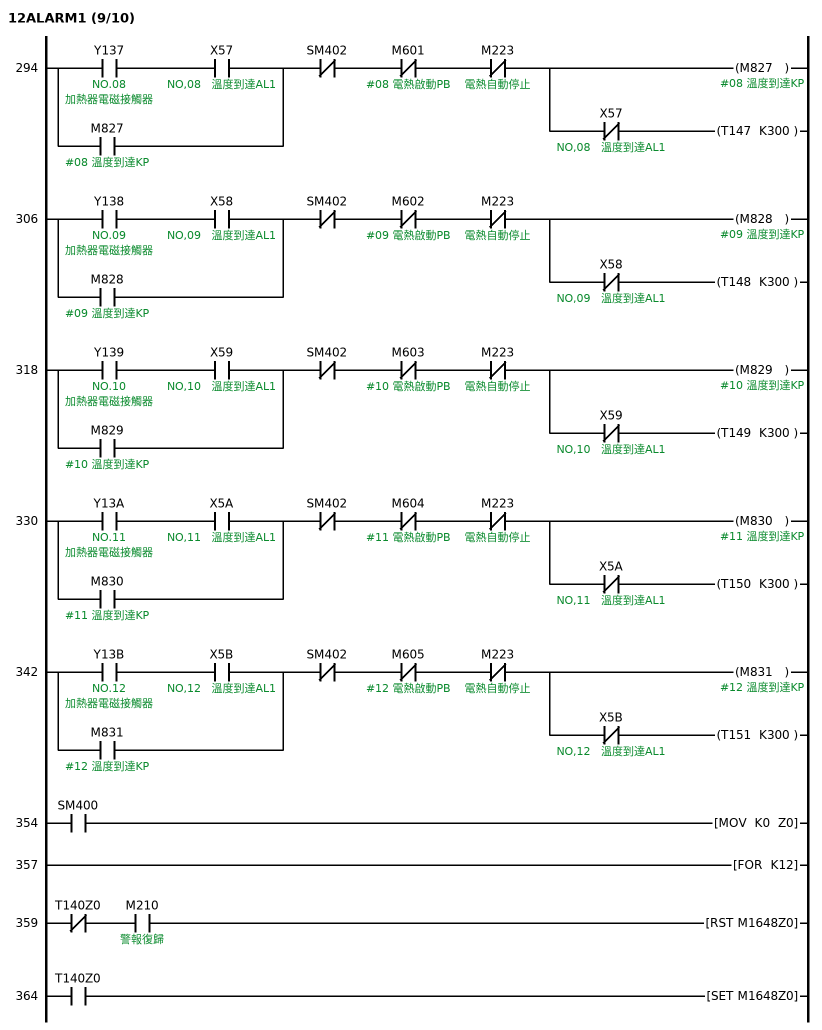
294   LD      Y137  ; NO.08   加熱器電磁接觸器
      AND     X57  ; NO,08   溫度到達AL1
      OR      M827  ; #08 溫度到達KP
      ANI     SM402
      ANI     M601  ; #08 電熱啟動PB
      ANI     M223  ; 電熱自動停止
      OUT     M827  ; #08 溫度到達KP
      ANI     X57  ; NO,08   溫度到達AL1
      OUT     T147 K300
306   LD      Y138  ; NO.09   加熱器電磁接觸器
      AND     X58  ; NO,09   溫度到達AL1
      OR      M828  ; #09 溫度到達KP
      ANI     SM402
      ANI     M602  ; #09 電熱啟動PB
      ANI     M223  ; 電熱自動停止
      OUT     M828  ; #09 溫度到達KP
      ANI     X58  ; NO,09   溫度到達AL1
      OUT     T148 K300
318   LD      Y139  ; NO.10   加熱器電磁接觸器
      AND     X59  ; NO,10   溫度到達AL1
      OR      M829  ; #10 溫度到達KP
      ANI     SM402
      ANI     M603  ; #10 電熱啟動PB
      ANI     M223  ; 電熱自動停止
      OUT     M829  ; #10 溫度到達KP
      ANI     X59  ; NO,10   溫度到達AL1
      OUT     T149 K300
330   LD      Y13A  ; NO.11   加熱器電磁接觸器
      AND     X5A  ; NO,11   溫度到達AL1
      OR      M830  ; #11 溫度到達KP
      ANI     SM402
      ANI     M604  ; #11 電熱啟動PB
      ANI     M223  ; 電熱自動停止
      OUT     M830  ; #11 溫度到達KP
      ANI     X5A  ; NO,11   溫度到達AL1
      OUT     T150 K300
342   LD      Y13B  ; NO.12   加熱器電磁接觸器
      AND     X5B  ; NO,12   溫度到達AL1
      OR      M831  ; #12 溫度到達KP
      ANI     SM402
      ANI     M605  ; #12 電熱啟動PB
      ANI     M223  ; 電熱自動停止
      OUT     M831  ; #12 溫度到達KP
      ANI     X5B  ; NO,12   溫度到達AL1
      OUT     T151 K300
354   LD      SM400
      MOV     K0 Z0
357   FOR     K12
359   LDI     T140Z0
      AND     M210  ; 警報復歸
      RST     M1648Z0
364   LD      T140Z0
      SET     M1648Z0
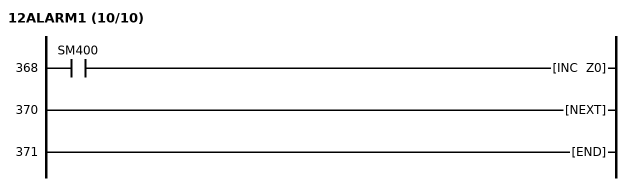
368   LD      SM400
      INC     Z0
370   NEXT
371   END
END_PROGRAM

PROGRAM 13ALARM2
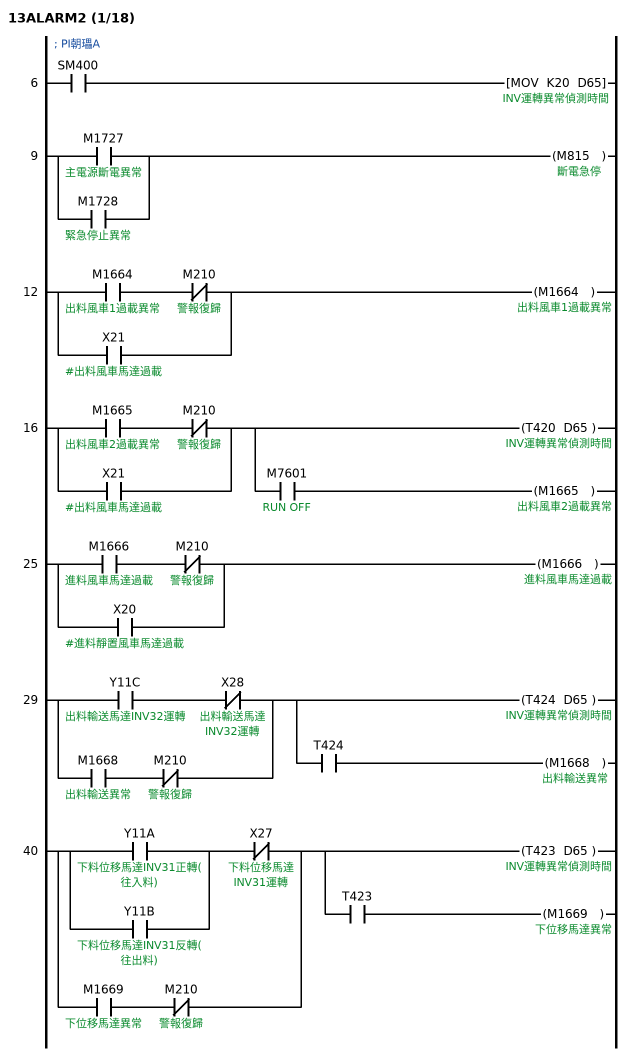
; PI朝瓃Α
6     LD      SM400
      MOV     K20 D65  ; INV運轉異常偵測時間
9     LD      M1727  ; 主電源斷電異常
      OR      M1728  ; 緊急停止異常
      OUT     M815  ; 斷電急停
12    LD      M1664  ; 出料風車1過載異常
      ANI     M210  ; 警報復歸
      OR      X21  ; #出料風車馬達過載
      OUT     M1664  ; 出料風車1過載異常
16    LD      M1665  ; 出料風車2過載異常
      ANI     M210  ; 警報復歸
      OR      X21  ; #出料風車馬達過載
      OUT     T420 D65  ; INV運轉異常偵測時間
      AND     M7601  ; RUN OFF
      OUT     M1665  ; 出料風車2過載異常
25    LD      M1666  ; 進料風車馬達過載
      ANI     M210  ; 警報復歸
      OR      X20  ; #進料靜置風車馬達過載
      OUT     M1666  ; 進料風車馬達過載
29    LD      Y11C  ; 出料輸送馬達INV32運轉
      ANI     X28  ; 出料輸送馬達    INV32運轉
      LD      M1668  ; 出料輸送異常
      ANI     M210  ; 警報復歸
      ORB
      OUT     T424 D65  ; INV運轉異常偵測時間
      AND     T424
      OUT     M1668  ; 出料輸送異常
40    LD      Y11A  ; 下料位移馬達INV31正轉(往入料)
      OR      Y11B  ; 下料位移馬達INV31反轉(往出料)
      ANI     X27  ; 下料位移馬達    INV31運轉
      LD      M1669  ; 下位移馬達異常
      ANI     M210  ; 警報復歸
      ORB
      OUT     T423 D65  ; INV運轉異常偵測時間
      AND     T423
      OUT     M1669  ; 下位移馬達異常
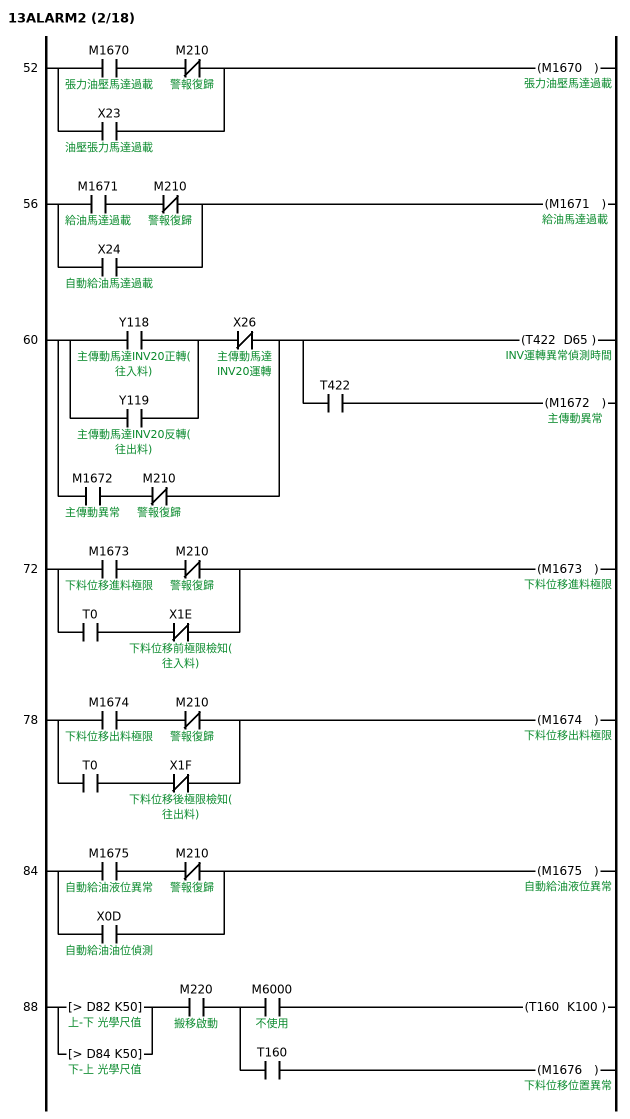
52    LD      M1670  ; 張力油壓馬達過載
      ANI     M210  ; 警報復歸
      OR      X23  ; 油壓張力馬達過載
      OUT     M1670  ; 張力油壓馬達過載
56    LD      M1671  ; 給油馬達過載
      ANI     M210  ; 警報復歸
      OR      X24  ; 自動給油馬達過載
      OUT     M1671  ; 給油馬達過載
60    LD      Y118  ; 主傳動馬達INV20正轉(往入料)
      OR      Y119  ; 主傳動馬達INV20反轉(往出料)
      ANI     X26  ; 主傳動馬達      INV20運轉
      LD      M1672  ; 主傳動異常
      ANI     M210  ; 警報復歸
      ORB
      OUT     T422 D65  ; INV運轉異常偵測時間
      AND     T422
      OUT     M1672  ; 主傳動異常
72    LD      M1673  ; 下料位移進料極限
      ANI     M210  ; 警報復歸
      LD      T0
      ANI     X1E  ; 下料位移前極限檢知(往入料)
      ORB
      OUT     M1673  ; 下料位移進料極限
78    LD      M1674  ; 下料位移出料極限
      ANI     M210  ; 警報復歸
      LD      T0
      ANI     X1F  ; 下料位移後極限檢知(往出料)
      ORB
      OUT     M1674  ; 下料位移出料極限
84    LD      M1675  ; 自動給油液位異常
      ANI     M210  ; 警報復歸
      OR      X0D  ; 自動給油油位偵測
      OUT     M1675  ; 自動給油液位異常
88    LD>     D82 K50  ; 上-下 光學尺值
      OR>     D84 K50  ; 下-上 光學尺值
      AND     M220  ; 搬移啟動
      MPS
      AND     M6000  ; 不使用
      OUT     T160 K100
      MPP
      AND     T160
      OUT     M1676  ; 下料位移位置異常
